# EPICS StreamDevice protocol: dg645App/Db/dg645.proto
InTerminator=CR LF;
OutTerminator=CR;
ReadTimeout=1500;

idn              { out "*idn?"                           ;in "%100c"                ; }
getStatus        { out "*stb?"                           ;in "%d"                   ; }
getErr           { out "lerr?"                           ;in "%d"                   ; }
getTimebase      { out "timb?"                           ;in "%d"                   ; }
getIPAddr        { out "ifcf? 11"                        ;in "%s"                   ; }

getTrigSrc       { out "tsrc?"                           ;in "%d"                   ; }
setTrigSrc       { out "tsrc %d"                                                    ; }
getTrigLvl       { out "tlvl?"                           ;in "%f"                   ; }
setTrigLvl       { out "tlvl %f"                                                    ; }
getTrigRate      { out "trat?"                           ;in "%f"                   ; }
setTrigRate      { out "trat %f"                                                    ; }
singleShot       { out "*trg"                                                       ; }

getBurstMode     { out "burm?"                           ;in "%d"                   ; }
getBurstCnt      { out "burc?"                           ;in "%d"                   ; }
getBurstDelay    { out "burd?"                           ;in "%f"                   ; }
getBurstPeriod   { out "burp?"                           ;in "%f"                   ; }

getAdvTrigMode   { out "advt?"                           ;in "%d"                   ; }
getTrigHoldoff   { out "hold?"                           ;in "%f"                   ; }
getTrigInhibit   { out "inhb?"                           ;in "%d"                   ; }

getDelay         { out "dlay? \$1"                       ;in "%*d,%f"               ; }
setDelay         { out "dlay  \$1,%(\$2)d,%e"                                       ; }
getRef           { out "link? \$1"                       ;in "%d"                   ; }
setRef           { out "link  \$1,%d"                                               ; }
